{attribute 'obsolete' := 'Use F_TaskTime - F_GetTaskTime conflicts with Tc2_System.F_GetTaskTime'}
FUNCTION F_GetTaskTime : LREAL
VAR
    TaskIndex : DINT;
END_VAR

TaskIndex := GETCURTASKINDEXEX();
IF TaskIndex > 0 THEN
    F_GetTaskTime := UDINT_TO_LREAL(TwinCAT_SystemInfoVarList._taskInfo[TaskIndex].CycleTime) * LREAL#1E-7;
END_IF

END_FUNCTION

(* stored: Version 1.1.0.1, ProductVersion 3.1.4024.12
   POU F_GetTaskTime: Id {3952241e-3b2b-43a8-982f-df54c9a9a7c8}, SpecialFunc None *)
